TYPE ST_ConveyorRecipe :
	STRUCT
		Axis : ST_MotionLinxAxisRecipe;
		
	END_STRUCT
END_TYPE

(* stored: Version 1.1.0.1, ProductVersion 3.1.4024.16
   DUT ST_ConveyorRecipe: Id {34034440-ba56-4868-a462-3a35490a3945} *)
